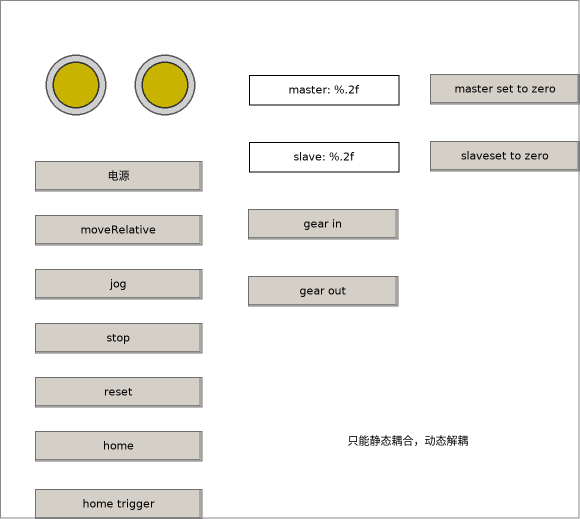
VISUALIZATION couple  // 580x519
    Lamp1 (41,50 70x70), variable: master.axis.NcToPlc.StateDWord.20, style: Lamp-Lamp1-Yellow
    Button (35,161 167x30), "电源"
        OnMouseClick: execute { master.shouldPowerOn := NOT master.shouldPowerOn; slave.shouldPowerOn := NOT slave.shouldPowerOn; }
    Lamp1 (130,50 70x70), variable: slave.axis.NcToPlc.StateDWord.20, style: Lamp-Lamp1-Yellow
    Rectangle (249,75 150x30), "master: %.2f", text variable: master.axis.NcToPlc.ActPos
    Rectangle (249,142 150x30), "slave: %.2f", text variable: slave.axis.NcToPlc.ActPos
    Button (35,215 167x30), "moveRelative"
        tap master.shouldMoveRel
    Button (35,269 167x30), "jog"
        OnMouseClick: execute { master.jogDirection := NOT master.jogDirection; master.shouldJog := TRUE; }
    Button (430,74 150x30), "master set to zero"
        tap master.shouldSetZero
    Button (35,323 167x30), "stop"
        tap master.shouldStop
    Button (35,377 167x30), "reset"
        tap master.shouldReset
    Button (430,141 150x30), "slaveset to zero"
        tap slave.shouldSetZero
    Button (248,209 150x30), "gear in"
        tap couple.shouldGearIn
    Button (248,276 150x30), "gear out"
        tap couple.shouldGearOut
    Button (35,431 167x30), "home"
        tap master.shouldGoHome
    Button (35,489 167x30), "home trigger"
        tap master.homeTrigger
    Label (333,426 150x30), "只能静态耦合，动态解耦"
END_VISUALIZATION

(* stored: Version 1.1.0.1, ProductVersion 3.1.4024.4
   Visu couple: Id {8f052f0f-85dd-421d-96f7-2dba2af33276} *)
